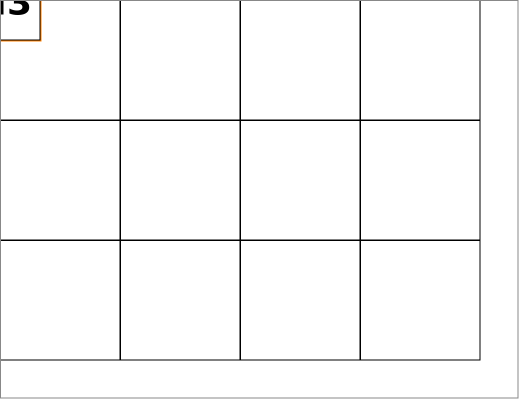
VISUALIZATION VI_Control_Xplanar  // 519x399
    Rectangle (0,0 120x120)
    Rectangle (120,0 120x120)
    Rectangle (240,0 120x120)
    Rectangle (360,0 120x120)
    Rectangle (0,120 120x120)
    Rectangle (120,120 120x120)
    Rectangle (240,120 120x120)
    Rectangle (360,120 120x120)
    Rectangle (0,240 120x120)
    Rectangle (120,240 120x120)
    Rectangle (240,240 120x120)
    Rectangle (360,240 120x120)
    Rectangle (-39,-39 80x80), "1"
        p3560616238: MAIN.fbXMotionUnit.fbStation_01_Process.VisuPosX/2
        p2738717112: (720-MAIN.fbXMotionUnit.fbStation_01_Process.VisuPosY)/2
    Rectangle (-39,-39 80x80), "2"
        p3560616238: MAIN.fbXMotionUnit.fbStation_02_Process.VisuPosX/2
        p2738717112: (720-MAIN.fbXMotionUnit.fbStation_02_Process.VisuPosY)/2
    Rectangle (-39,-39 80x80), "3"
        p3560616238: MAIN.fbXMotionUnit.fbStation_03_Process.VisuPosX/2
        p2738717112: (720-MAIN.fbXMotionUnit.fbStation_03_Process.VisuPosY)/2
    Rectangle (-39,-39 80x80), "4"
        p3560616238: MAIN.fbXMotionUnit.fbStation_04_Switch.VisuPosX/2
        p2738717112: (720-MAIN.fbXMotionUnit.fbStation_04_Switch.VisuPosY)/2
    Rectangle (-39,-39 80x80), "5"
        p3560616238: MAIN.fbXMotionUnit.fbStation_05_Switch.VisuPosX/2
        p2738717112: (720-MAIN.fbXMotionUnit.fbStation_05_Switch.VisuPosY)/2
    Rectangle (-37,-37 77x77), "M1"
        p3560616238: MAIN.fbXMotionUnit.fbMover[1].VisuPos.x/2
        p2738717112: (720-MAIN.fbXMotionUnit.fbMover[1].VisuPos.y)/2
    Rectangle (-37,-37 77x77), "M2"
        p3560616238: MAIN.fbXMotionUnit.fbMover[2].VisuPos.x/2
        p2738717112: (720-MAIN.fbXMotionUnit.fbMover[2].VisuPos.y)/2
    Rectangle (-37,-37 77x77), "M4"
        p3560616238: MAIN.fbXMotionUnit.fbMover[4].VisuPos.x/2
        p2738717112: (720-MAIN.fbXMotionUnit.fbMover[4].VisuPos.y)/2
    Rectangle (-37,-37 77x77), "M3"
        p3560616238: MAIN.fbXMotionUnit.fbMover[3].VisuPos.x/2
        p2738717112: (720-MAIN.fbXMotionUnit.fbMover[3].VisuPos.y)/2
END_VISUALIZATION

(* stored: Version 1.1.0.1, ProductVersion 3.1.4024.9
   Visu VI_Control_Xplanar: Id {ee1f2643-fbba-45a7-8b89-caf09ac9a565} *)
